{attribute 'qualified_only'}
{attribute 'strict'}
TYPE eEntryType :
(
	IntegerValue		:=	0,
	FloatValue			:=	1,
	StringValue			:=	2
);
END_TYPE

(* stored: Version 1.1.0.1, ProductVersion 3.1.4026.18
   DUT eEntryType: Id {84eab79a-e1bc-4d62-9b5c-220cfad47f20} *)
